TEXTLIST tlSensorNames
  0 = 'Bottle Sensor' | EN: 'Bottle Sensor' | PL: 'Bottle Sensor'
  1 = 'Bottle Eject Sensor' | EN: 'Bottle Eject Sensor' | PL: 'Bottle Eject Sensor'
   = ''
END_TEXTLIST

(* stored: Version 1.1.0.1, ProductVersion 3.1.4024.15
   TextList tlSensorNames: Id {09652da2-fae6-49b9-9b2a-10e94f8e2354} *)
